PROGRAM MAIN
VAR
	init : INT := 0;
	flag : INT := 0;
END_VAR

VAR_INPUT
	bmanual : BOOL;
	bPowerDisable: BOOL;
	bReadDone : BOOL;
END_VAR

HMILogic();
LoadModel();

Run.A_AlwaysActive();

IF bPowerDisable THEN
	Run.A_EnableManualMovement();
	Run.nManual := 0;
	flag := 0;
END_IF

IF bmanual THEN
	Run.A_ReadXYZValue();
	bReadDone := TRUE;
	
END_IF

IF HMILogic.bRun THEN
	IF flag = 0 THEN
		Run.A_EnableManualMovement();
		flag := flag + 1;
	END_IF
	Run(arrangedFrames := HMILogic.ArrangedFrames);
END_IF

END_PROGRAM

(* stored: Version 1.1.0.1, ProductVersion 3.1.4024.9
   POU MAIN: Id {6f26785d-3141-4d83-8f28-dd4e0f083bd8}, SpecialFunc None *)
